{attribute 'qualified_only'}
{attribute 'strict'}
TYPE EStopStatus:
(
        UNKNOWN := 0, 
		ENGAGED := 1, 
		DISENGAGED := 2
);
END_TYPE

(* stored: Version 1.1.0.1, ProductVersion 3.1.4024.12
   DUT EStopStatus: Id {a7105928-debf-494b-ac49-73fd12eb7476} *)
